RoboDK station: full) scene.rdk

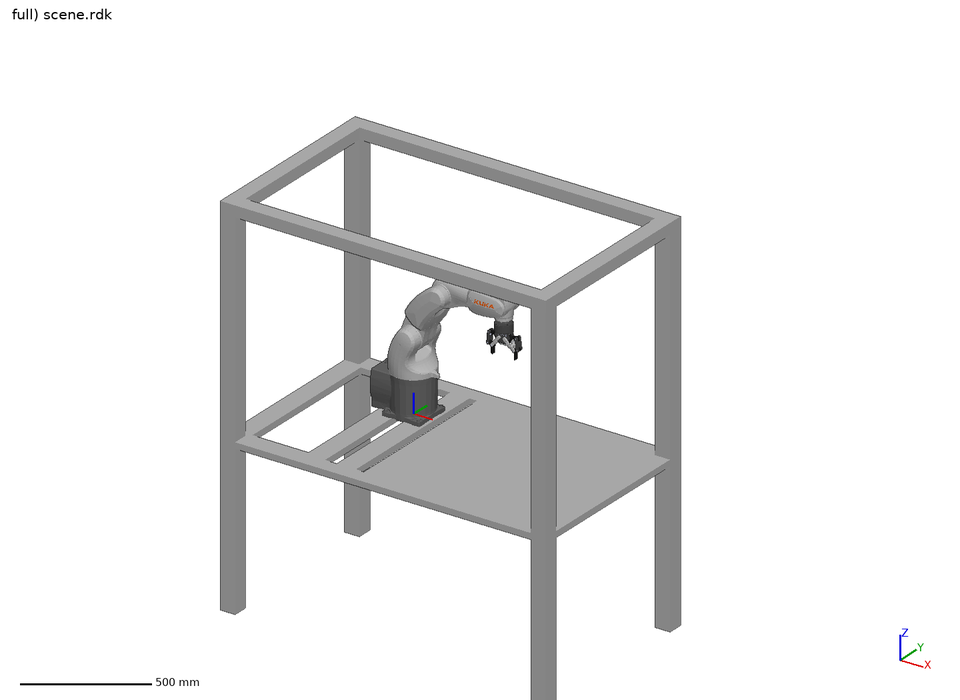
[picture v0: the station drawn from its stored meshes, robots at their saved joint values, targets as dots, program paths as lines]
Station full) scene. Poses are relative to the parent item; angles as X-Y-Z fixed-axis rotations.
  - frame KUKA KR 3 R540 Base at (-292.39, 11.5, 0) mm
    - robot KUKA KR 3 R540: 6 axes, payload 3 kg, reach 541 mm, repeatability 0.02 mm, weight 26 kg
        modified DH rows (alpha deg, a mm, theta deg, d mm): 0, 0, 0, 345; -90, 20, 0, 0; 0, 260, -90, 0; -90, 20, 0, 260; 90, 0, 0, 0; -90, 0, 180, 75
        joint limits [-170, -170, -110, -175, -120, -350] to [170, 50, 155, 175, 120, 350]; home [0, -90, 90, 0, 0, 0]; saved at [1, -57, 57, 0, 89, 2.16]
      - tool Gripper RobotiQ 85 Opened, TCP at (0, -20, 130) mm, size 147.4 x 146.8 x 75 mm
  - object  at (736.15, -583.05, -13.07) mm, rotated rx 0 ry 0 rz 90 deg, size 107739.4 x 3125.1 x 1726.8 mm, geometry from  v2.stl
